(* IEC 61131-3 sources: repolevel_ST_code_completion/output/full_case_fixed/repoeval_open-type_dual-axis_winding_machine/readful_result_history, 17 files *)

(* ---- F_CalculateRadius_0.st ---- *)
FUNCTION F_CalculateRadius : LREAL
VAR_INPUT
	lD				:	LREAL;		//两轴中心距离
	lHold			:	LREAL;		//测量开始时的AxisV位置
	lHnew			:	LREAL;		//测量结束时的AxisV位置
	lTk				:	LREAL;		//材料厚度
	lOffset			:	LREAL;		//高度偏移量
END_VAR
VAR
    lRadiusStart : LREAL;
    lRadiusEnd : LREAL;
    lResult : LREAL;
END_VAR

lRadiusStart := SQRT(EXPT(lD, 2) + EXPT(lHold + lOffset, 2));
lRadiusEnd := SQRT(EXPT(lD, 2) + EXPT(lHnew + lOffset, 2));
lResult := ABS(lRadiusEnd - lRadiusStart) / SMC_PI + lTk;

F_CalculateRadius := lResult;
RETURN;
END_FUNCTION

(* ---- F_CalculateRadius_1.st ---- *)
FUNCTION F_CalculateRadius : LREAL
VAR_INPUT
	lD				:	LREAL;		//两轴中心距离
	lHold			:	LREAL;		//测量开始时的AxisV位置
	lHnew			:	LREAL;		//测量结束时的AxisV位置
	lTk				:	LREAL;		//材料厚度
	lOffset			:	LREAL;		//高度偏移量
END_VAR
VAR
    lRadiusStart : LREAL;
    lRadiusEnd : LREAL;
    lResult : LREAL;
END_VAR

lRadiusStart := SQRT(POW(lD, 2) + POW(lHold + lOffset, 2));
lRadiusEnd := SQRT(POW(lD, 2) + POW(lHnew + lOffset, 2));
lResult := ABS(lRadiusEnd - lRadiusStart) / PI + lTk;

F_CalculateRadius := lResult;
RETURN;
END_FUNCTION

(* ---- F_CompensateVelocity_0.st ---- *)
FUNCTION F_CompensateVelocity : LREAL
VAR_INPUT
	lCurrentVel		:	LREAL;		//当前速度
	lOldPos			:	LREAL;		//上一次位置
	lNewPos			:	LREAL;		//当前位置
	lRadius			:	LREAL;		//当前半径
	lTk				:	LREAL;		//材料厚度
	bUnwinding		:	BOOL;		//TRUE=放卷（半径减小），FALSE=收卷（半径增加）
END_VAR
VAR
    lDeltaPos : LREAL; // Position change
END_VAR

// Calculate position change
lDeltaPos := lNewPos - lOldPos;

// Check if the axis is moving (position change)
IF lDeltaPos <> 0 THEN
    IF bUnwinding THEN
        // Unwinding: radius decreases, velocity needs to increase
        // Formula: V_new = V_old + V_old * Tk / (R - Tk)
        IF (lRadius - lTk) > 0.01 THEN // Avoid division by zero
            F_CompensateVelocity := lCurrentVel + lCurrentVel * lTk / (lRadius - lTk);
        ELSE
            F_CompensateVelocity := lCurrentVel;
        END_IF
    ELSE
        // Rewinding: radius increases, velocity needs to decrease
        // Formula: V_new = V_old - V_old * Tk / (R + Tk)
        IF (lRadius + lTk) > 0.01 THEN // Avoid division by zero
            F_CompensateVelocity := lCurrentVel - lCurrentVel * lTk / (lRadius + lTk);
        ELSE
            F_CompensateVelocity := lCurrentVel;
        END_IF
    END_IF
ELSE
    // Position unchanged, maintain current velocity
    F_CompensateVelocity := lCurrentVel;
END_IF;

RETURN;
END_FUNCTION

(* ---- F_CompensateVelocity_1.st ---- *)
FUNCTION F_CompensateVelocity : LREAL
VAR_INPUT
  lCurrentVel		:	LREAL;		//当前速度
  lOldPos			:	LREAL;		//上一次位置
  lNewPos			:	LREAL;		//当前位置
  lRadius			:	LREAL;		//当前半径
  lTk				:	LREAL;		//材料厚度
  bUnwinding		:	BOOL;		//TRUE=放卷（半径减小），FALSE=收卷（半径增加）
END_VAR
VAR
  lDeltaPos : LREAL; // Position change
END_VAR

// Calculate position change
lDeltaPos := lNewPos - lOldPos;

// Check if the axis is moving (position change)
IF lDeltaPos <> 0 THEN
  IF bUnwinding THEN
    // Unwinding: radius decreases, velocity needs to increase
    // Formula: V_new = V_old + V_old * Tk / (R - Tk)
    IF (lRadius - lTk) > 0.01 THEN // Avoid division by zero
      F_CompensateVelocity := lCurrentVel + lCurrentVel * lTk / (lRadius - lTk);
    ELSE
      F_CompensateVelocity := lCurrentVel;
    END_IF
  ELSE
    // Rewinding: radius increases, velocity needs to decrease
    // Formula: V_new = V_old - V_old * Tk / (R + Tk)
    IF (lRadius + lTk) > 0.01 THEN // Avoid division by zero
      F_CompensateVelocity := lCurrentVel - lCurrentVel * lTk / (lRadius + lTk);
    ELSE
      F_CompensateVelocity := lCurrentVel;
    END_IF
  END_IF
ELSE
  // Position unchanged, maintain current velocity
  F_CompensateVelocity := lCurrentVel;
END_IF;

RETURN;
END_FUNCTION

(* ---- F_CompensateVelocity_2.st ---- *)
FUNCTION F_CompensateVelocity : LREAL
VAR_INPUT
 lCurrentVel		:	LREAL;		//当前速度
 lOldPos			:	LREAL;		//上一次位置
 lNewPos			:	LREAL;		//当前位置
 lRadius			:	LREAL;		//当前半径
 lTk				:	LREAL;		//材料厚度
 bUnwinding		:	BOOL;		//TRUE=放卷（半径减小），FALSE=收卷（半径增加）
END_VAR
VAR
 lDeltaPos : LREAL; // Position change
END_VAR

// Calculate position change
lDeltaPos := lNewPos - lOldPos;

// Check if the axis is moving (position change)
IF lDeltaPos <> 0 THEN
 IF bUnwinding THEN
  // Unwinding: radius decreases, velocity needs to increase
  // Formula: V_new = V_old + V_old * Tk / (R - Tk)
  IF (lRadius - lTk) > 0.01 THEN // Avoid division by zero
   F_CompensateVelocity := lCurrentVel + lCurrentVel * lTk / (lRadius - lTk);
  ELSE
   F_CompensateVelocity := lCurrentVel;
  END_IF
 ELSE
  // Rewinding: radius increases, velocity needs to decrease
  // Formula: V_new = V_old - V_old * Tk / (R + Tk)
  IF (lRadius + lTk) > 0.01 THEN // Avoid division by zero
   F_CompensateVelocity := lCurrentVel - lCurrentVel * lTk / (lRadius + lTk);
  ELSE
   F_CompensateVelocity := lCurrentVel;
  END_IF
 END_IF
ELSE
 // Position unchanged, maintain current velocity
 F_CompensateVelocity := lCurrentVel;
END_IF;

RETURN;
END_FUNCTION

(* ---- F_CompensateVelocity_3.st ---- *)
FUNCTION F_CompensateVelocity : LREAL
VAR_INPUT
lCurrentVel		:	LREAL;		//当前速度
lOldPos			:	LREAL;		//上一次位置
lNewPos			:	LREAL;		//当前位置
lRadius			:	LREAL;		//当前半径
lTk				:	LREAL;		//材料厚度
bUnwinding		:	BOOL;		//TRUE=放卷（半径减小），FALSE=收卷（半径增加）
END_VAR
VAR
lDeltaPos : LREAL; // Position change
END_VAR

// Calculate position change
lDeltaPos := lNewPos - lOldPos;

// Check if the axis is moving (position change)
IF lDeltaPos <> 0 THEN
IF bUnwinding THEN
 // Unwinding: radius decreases, velocity needs to increase
 // Formula: V_new = V_old + V_old * Tk / (R - Tk)
 IF (lRadius - lTk) > 0.01 THEN // Avoid division by zero
 F_CompensateVelocity := lCurrentVel + lCurrentVel * lTk / (lRadius - lTk);
 ELSE
 F_CompensateVelocity := lCurrentVel;
 END_IF
ELSE
 // Rewinding: radius increases, velocity needs to decrease
 // Formula: V_new = V_old - V_old * Tk / (R + Tk)
 IF (lRadius + lTk) > 0.01 THEN // Avoid division by zero
 F_CompensateVelocity := lCurrentVel - lCurrentVel * lTk / (lRadius + lTk);
 ELSE
 F_CompensateVelocity := lCurrentVel;
 END_IF
END_IF
ELSE
// Position unchanged, maintain current velocity
F_CompensateVelocity := lCurrentVel;
END_IF;

RETURN;
END_FUNCTION

(* ---- CheckF_0.st ---- *)
FUNCTION_BLOCK CheckF
VAR_INPUT
	lM	:	LREAL;
	lL	:	LREAL;
	lH	:	LREAL;
END_VAR
VAR_OUTPUT
	lF	:	LREAL;
END_VAR
VAR
END_VAR

IF lH <> 0 THEN
    lF := 9.8 * lM / (2 * COS(ATAN(lL / lH)));
ELSE
    lF := 0;
END_IF
END_FUNCTION_BLOCK

(* ---- CheckF_1.st ---- *)
FUNCTION_BLOCK CheckF
VAR_INPUT
	lM	:	LREAL;
	lL	:	LREAL;
	lH	:	LREAL;
END_VAR
VAR_OUTPUT
	lF	:	LREAL;
END_VAR
VAR
END_VAR

IF lH <> 0 THEN
  lF := 9.8 * lM / (2 * COS(ATAN(REAL(lL / lH))));
ELSE
  lF := 0;
END_IF
END_FUNCTION_BLOCK

(* ---- CheckF_2.st ---- *)
FUNCTION_BLOCK CheckF
VAR_INPUT
	lM	:	LREAL;
	lL	:	LREAL;
	lH	:	LREAL;
END_VAR
VAR_OUTPUT
	lF	:	LREAL;
END_VAR
VAR
END_VAR

IF lH <> 0 THEN
 lF := 9.8 * lM / (2 * COS(ATAN(REAL(lL) / REAL(lH))));
ELSE
 lF := 0;
END_IF
END_FUNCTION_BLOCK

(* ---- CheckF_3.st ---- *)
FUNCTION_BLOCK CheckF
VAR_INPUT
	lM	:	LREAL;
	lL	:	LREAL;
	lH	:	LREAL;
END_VAR
VAR_OUTPUT
	lF	:	LREAL;
END_VAR
VAR
END_VAR

IF lH <> 0 THEN
lF := LREAL(9.8 * lM / (2 * COS(ATAN(REAL(lL) / REAL(lH)))));
ELSE
lF := 0;
END_IF
END_FUNCTION_BLOCK

(* ---- SeekHome_0.st ---- *)
FUNCTION_BLOCK SeekHome
VAR_IN_OUT
	_Axis	:	AXIS_REF_SM3;
END_VAR
VAR_INPUT
	_xHome	:	BOOL;
	_xAbort	:	BOOL;
	_nHomeMode	:	HomeMode;
	_fFastHomeVel	:	LREAL;
	_fSlowHomeVel	:	LREAL;
	_fHomeAcc		:	LREAL;
	_fHomeDec		:	LREAL;
	_fHomePos		:	LREAL;
	_xReferenceSwitch	:	BOOL;//typically is true
	_nDirection	:	MC_DIRECTION;
	_xIndexPulse	:	BOOL;
END_VAR
VAR_OUTPUT
	_xBusy	:	BOOL;
	_xDone	:	BOOL;
	_xErr	:	BOOL;
	_iErrId	:	DINT;
END_VAR
VAR
    _fbMoveVel : MC_MoveVelocity;
    _fbMoveAbs : MC_MoveAbsolute;
    _fbHalt : MC_Halt;
    _fbSetPos : MC_SetPosition;
    _fbRtrig : R_TRIG;
    _fbFtrig : F_TRIG;
    _nBDirection : MC_DIRECTION;
    _fTempPos : LREAL;
    _nState : USINT;
    _xPrevHome : BOOL;
END_VAR

CASE _nState OF
    0: // Idle state
        _xBusy := FALSE;
        _xDone := FALSE;
        _xErr := FALSE;
        _iErrId := 0;
        IF _xHome THEN
            _xBusy := TRUE;
            _nState := 1;
        END_IF;

    1: // Start homing sequence
        _fbMoveVel.Execute := TRUE;
        _fbMoveVel.Axis := _Axis;
        _fbMoveVel.Velocity := _fFastHomeVel;
        _fbMoveVel.Acceleration := _fHomeAcc;
        _fbMoveVel.Deceleration := _fHomeDec;
        _fbMoveVel.Direction := _nDirection;

        IF _fbMoveVel.Error THEN
            _xErr := TRUE;
            _iErrId := _fbMoveVel.ErrorID;
            _fbMoveVel.Execute := FALSE;
            _nState := 0;
        ELSIF _xReferenceSwitch THEN
            _fbMoveVel.Execute := FALSE;
            _nState := 2;
        END_IF;

    2: // Slow homing
        _fbMoveVel.Execute := TRUE;
        _fbMoveVel.Axis := _Axis;
        _fbMoveVel.Velocity := _fSlowHomeVel;
        _fbMoveVel.Acceleration := _fHomeAcc;
        _fbMoveVel.Deceleration := _fHomeDec;
        _fbMoveVel.Direction := _nDirection;

        IF _fbMoveVel.Error THEN
            _xErr := TRUE;
            _iErrId := _fbMoveVel.ErrorID;
            _fbMoveVel.Execute := FALSE;
            _nState := 0;
        ELSIF _xIndexPulse THEN
            _fbMoveVel.Execute := FALSE;
            _nState := 3;
        END_IF;

    3: // Set position
        _fbSetPos.Execute := TRUE;
        _fbSetPos.Axis := _Axis;
        _fbSetPos.Position := _fHomePos;

        IF _fbSetPos.Error THEN
            _xErr := TRUE;
            _iErrId := _fbSetPos.ErrorID;
            _fbSetPos.Execute := FALSE;
            _nState := 0;
        ELSIF _fbSetPos.Done THEN
            _fbSetPos.Execute := FALSE;
            _nState := 4;
        END_IF;

    4: // Homing complete
        _xBusy := FALSE;
        _xDone := TRUE;
        _nState := 0;

END_CASE;

IF _xAbort THEN
    _fbMoveVel.Execute := FALSE;
    _fbSetPos.Execute := FALSE;
    _xBusy := FALSE;
    _xDone := FALSE;
    _xErr := FALSE;
    _iErrId := 0;
    _nState := 0;
END_IF;
END_FUNCTION_BLOCK

(* ---- SeekHome_2.st ---- *)
FUNCTION_BLOCK SeekHome
VAR_IN_OUT
	_Axis	:	AXIS_REF_SM3;
END_VAR
VAR_INPUT
	_xHome	:	BOOL;
	_xAbort	:	BOOL;
	_nHomeMode	:	HomeMode;
	_fFastHomeVel	:	LREAL;
	_fSlowHomeVel	:	LREAL;
	_fHomeAcc		:	LREAL;
	_fHomeDec		:	LREAL;
	_fHomePos		:	LREAL;
	_xReferenceSwitch	:	BOOL;//typically is true
	_nDirection	:	MC_DIRECTION;
	_xIndexPulse	:	BOOL;
END_VAR
VAR_OUTPUT
	_xBusy	:	BOOL;
	_xDone	:	BOOL;
	_xErr	:	BOOL;
	_iErrId	:	DINT;
END_VAR
VAR
    _fbMoveVel : MC_MoveVelocity;
    _fbMoveAbs : MC_MoveAbsolute;
    _fbHalt : MC_Halt;
    _fbSetPos : MC_SetPosition;
    _fbRtrig : R_TRIG;
    _fbFtrig : F_TRIG;
    _nBDirection : MC_DIRECTION;
    _fTempPos : LREAL;
    _nState : USINT;
    _xPrevHome : BOOL;
END_VAR

CASE _nState OF
    0: // Idle state
        _xBusy := FALSE;
        _xDone := FALSE;
        _xErr := FALSE;
        _iErrId := 0;
        IF _xHome THEN
            _xBusy := TRUE;
            _nState := 1;
        END_IF;

    1: // Start homing sequence
_fbMoveVel.Axis := _Axis;
    _fbMoveVel.Velocity := _fFastHomeVel;
    _fbMoveVel.Acceleration := _fHomeAcc;
    _fbMoveVel.Deceleration := _fHomeDec;
    _fbMoveVel.Direction := _nDirection;

    IF NOT _fbMoveVel.Enabled THEN
      _fbMoveVel.Execute := TRUE;
    END_IF;

    IF _fbMoveVel.Error THEN
      _xErr := TRUE;
      _iErrId := _fbMoveVel.ErrorID;
      _fbMoveVel.Execute := FALSE;
      _nState := 0;
    ELSIF _xReferenceSwitch THEN
      _fbMoveVel.Execute := FALSE;
      _nState := 2;
    END_IF;

    2: // Slow homing
_fbMoveVel.Axis := _Axis;
    _fbMoveVel.Velocity := _fSlowHomeVel;
    _fbMoveVel.Acceleration := _fHomeAcc;
    _fbMoveVel.Deceleration := _fHomeDec;
    _fbMoveVel.Direction := _nDirection;

    IF NOT _fbMoveVel.Enabled THEN
      _fbMoveVel.Execute := TRUE;
    END_IF;

    IF _fbMoveVel.Error THEN
      _xErr := TRUE;
      _iErrId := _fbMoveVel.ErrorID;
      _fbMoveVel.Execute := FALSE;
      _nState := 0;
    ELSIF _xIndexPulse THEN
      _fbMoveVel.Execute := FALSE;
      _nState := 3;
    END_IF;

    3: // Set position
_fbSetPos.Axis := _Axis;
    _fbSetPos.Position := _fHomePos;

    IF NOT _fbSetPos.Enabled THEN
      _fbSetPos.Execute := TRUE;
    END_IF;

    IF _fbSetPos.Error THEN
      _xErr := TRUE;
      _iErrId := _fbSetPos.ErrorID;
      _fbSetPos.Execute := FALSE;
      _nState := 0;
    ELSIF _fbSetPos.Done THEN
      _fbSetPos.Execute := FALSE;
      _nState := 4;
    END_IF;

    4: // Homing complete
        _xBusy := FALSE;
        _xDone := TRUE;
        _nState := 0;

END_CASE;

IF _xAbort THEN
    _fbMoveVel.Execute := FALSE;
    _fbSetPos.Execute := FALSE;
    _xBusy := FALSE;
    _xDone := FALSE;
    _xErr := FALSE;
    _iErrId := 0;
    _nState := 0;
END_IF;
END_FUNCTION_BLOCK

(* ---- SeekHome_3.st ---- *)
FUNCTION_BLOCK SeekHome
VAR_IN_OUT
	_Axis	:	AXIS_REF_SM3;
END_VAR
VAR_INPUT
	_xHome	:	BOOL;
	_xAbort	:	BOOL;
	_nHomeMode	:	HomeMode;
	_fFastHomeVel	:	LREAL;
	_fSlowHomeVel	:	LREAL;
	_fHomeAcc		:	LREAL;
	_fHomeDec		:	LREAL;
	_fHomePos		:	LREAL;
	_xReferenceSwitch	:	BOOL;//typically is true
	_nDirection	:	MC_DIRECTION;
	_xIndexPulse	:	BOOL;
END_VAR
VAR_OUTPUT
	_xBusy	:	BOOL;
	_xDone	:	BOOL;
	_xErr	:	BOOL;
	_iErrId	:	DINT;
END_VAR
VAR
    _fbMoveVel : MC_MoveVelocity;
    _fbMoveAbs : MC_MoveAbsolute;
    _fbHalt : MC_Halt;
    _fbSetPos : MC_SetPosition;
    _fbRtrig : R_TRIG;
    _fbFtrig : F_TRIG;
    _nBDirection : MC_DIRECTION;
    _fTempPos : LREAL;
    _nState : USINT;
    _xPrevHome : BOOL;
END_VAR

CASE _nState OF
    0: // Idle state
        _xBusy := FALSE;
        _xDone := FALSE;
        _xErr := FALSE;
        _iErrId := 0;
        IF _xHome THEN
            _xBusy := TRUE;
            _nState := 1;
        END_IF;

    1: // Start homing sequence
_fbMoveVel.Axis := _Axis;
  _fbMoveVel.Velocity := _fFastHomeVel;
  _fbMoveVel.Acceleration := _fHomeAcc;
  _fbMoveVel.Deceleration := _fHomeDec;
  _fbMoveVel.Direction := _nDirection;

IF NOT _fbMoveVel.Execute THEN
   _fbMoveVel.Execute := TRUE;
  END_IF;

    IF _fbMoveVel.Error THEN
      _xErr := TRUE;
      _iErrId := _fbMoveVel.ErrorID;
      _fbMoveVel.Execute := FALSE;
      _nState := 0;
    ELSIF _xReferenceSwitch THEN
      _fbMoveVel.Execute := FALSE;
      _nState := 2;
    END_IF;

    2: // Slow homing
_fbMoveVel.Axis := _Axis;
  _fbMoveVel.Velocity := _fSlowHomeVel;
  _fbMoveVel.Acceleration := _fHomeAcc;
  _fbMoveVel.Deceleration := _fHomeDec;
  _fbMoveVel.Direction := _nDirection;

    IF NOT _fbMoveVel.Enabled THEN
      _fbMoveVel.Execute := TRUE;
    END_IF;

    IF _fbMoveVel.Error THEN
      _xErr := TRUE;
      _iErrId := _fbMoveVel.ErrorID;
      _fbMoveVel.Execute := FALSE;
      _nState := 0;
    ELSIF _xIndexPulse THEN
      _fbMoveVel.Execute := FALSE;
      _nState := 3;
    END_IF;

    3: // Set position
_fbSetPos.Axis := _Axis;
    _fbSetPos.Position := _fHomePos;

IF NOT _fbSetPos.Execute THEN
   _fbSetPos.Execute := TRUE;
  END_IF;

    IF _fbSetPos.Error THEN
      _xErr := TRUE;
      _iErrId := _fbSetPos.ErrorID;
      _fbSetPos.Execute := FALSE;
      _nState := 0;
    ELSIF _fbSetPos.Done THEN
      _fbSetPos.Execute := FALSE;
      _nState := 4;
    END_IF;

    4: // Homing complete
        _xBusy := FALSE;
        _xDone := TRUE;
        _nState := 0;

END_CASE;

IF _xAbort THEN
    _fbMoveVel.Execute := FALSE;
    _fbSetPos.Execute := FALSE;
    _xBusy := FALSE;
    _xDone := FALSE;
    _xErr := FALSE;
    _iErrId := 0;
    _nState := 0;
END_IF;
END_FUNCTION_BLOCK

(* ---- StaDisplay_0.st ---- *)
FUNCTION_BLOCK StaDisplay
VAR_INPUT
	iStatus :	INT;
END_VAR
VAR_OUTPUT
	Y1,Y2,Y3,Y4,Y5,Y6	:	BOOL;
END_VAR
VAR
END_VAR

CASE iStatus OF
    2,3,4,5,6,7,8,9,10,221,222:
        Y5 := FALSE;
        Y6 := TRUE;
        Y1 := TRUE;
        Y2 := FALSE;
        Y3 := FALSE;
        Y4 := FALSE;
    11,12:
        Y5 := FALSE;
        Y6 := TRUE;
        Y1 := FALSE;
        Y2 := TRUE;
        Y3 := FALSE;
        Y4 := FALSE;
    13,14,15,16,17,18,19,20,21,22:
        Y5 := TRUE;
        Y6 := FALSE;
        Y1 := FALSE;
        Y2 := FALSE;
        Y3 := TRUE;
        Y4 := FALSE;
    23,24:
        Y5 := TRUE;
        Y6 := FALSE;
        Y1 := FALSE;
        Y2 := FALSE;
        Y3 := FALSE;
        Y4 := TRUE;
    ELSE
        Y5 := FALSE;
        Y6 := FALSE;
        Y1 := FALSE;
        Y2 := FALSE;
        Y3 := FALSE;
        Y4 := FALSE;
END_CASE;
END_FUNCTION_BLOCK

(* ---- StaDisplay_1.st ---- *)
FUNCTION_BLOCK StaDisplay
VAR_INPUT
	iStatus :	INT;
END_VAR
VAR_OUTPUT
	Y1,Y2,Y3,Y4,Y5,Y6	:	BOOL;
END_VAR
VAR

END_VAR

CASE iStatus OF
  2,3,4,5,6,7,8,9,10,221,222:
    Y5 := FALSE;
    Y6 := TRUE;
    Y1 := TRUE;
    Y2 := FALSE;
    Y3 := FALSE;
    Y4 := FALSE;
  11,12:
    Y5 := FALSE;
    Y6 := TRUE;
    Y1 := FALSE;
    Y2 := TRUE;
    Y3 := FALSE;
    Y4 := FALSE;
  13,14,15,16,17,18,19,20,21,22:
    Y5 := TRUE;
    Y6 := FALSE;
    Y1 := FALSE;
    Y2 := FALSE;
    Y3 := TRUE;
    Y4 := FALSE;
  23,24:
    Y5 := TRUE;
    Y6 := FALSE;
    Y1 := FALSE;
    Y2 := FALSE;
    Y3 := FALSE;
    Y4 := TRUE;
  ELSE
    Y5 := FALSE;
    Y6 := FALSE;
    Y1 := FALSE;
    Y2 := FALSE;
    Y3 := FALSE;
    Y4 := FALSE;
END_CASE;
END_FUNCTION_BLOCK

(* ---- StaDisplay_2.st ---- *)
FUNCTION_BLOCK StaDisplay
VAR_INPUT
	iStatus :	INT;
END_VAR
VAR_OUTPUT
	Y1,Y2,Y3,Y4,Y5,Y6	:	BOOL;
END_VAR
CASE iStatus OF
 2,3,4,5,6,7,8,9,10,221,222:
  Y5 := FALSE;
  Y6 := TRUE;
  Y1 := TRUE;
  Y2 := FALSE;
  Y3 := FALSE;
  Y4 := FALSE;
 11,12:
  Y5 := FALSE;
  Y6 := TRUE;
  Y1 := FALSE;
  Y2 := TRUE;
  Y3 := FALSE;
  Y4 := FALSE;
 13,14,15,16,17,18,19,20,21,22:
  Y5 := TRUE;
  Y6 := FALSE;
  Y1 := FALSE;
  Y2 := FALSE;
  Y3 := TRUE;
  Y4 := FALSE;
 23,24:
  Y5 := TRUE;
  Y6 := FALSE;
  Y1 := FALSE;
  Y2 := FALSE;
  Y3 := FALSE;
  Y4 := TRUE;
 ELSE
  Y5 := FALSE;
  Y6 := FALSE;
  Y1 := FALSE;
  Y2 := FALSE;
  Y3 := FALSE;
  Y4 := FALSE;
END_CASE;
END_FUNCTION_BLOCK

(* ---- StaDisplay_3.st ---- *)
FUNCTION_BLOCK StaDisplay
VAR_INPUT
	iStatus :	INT;
END_VAR
VAR_OUTPUT
  Y1,Y2,Y3,Y4,Y5,Y6	:	BOOL;
END_VAR

CASE iStatus OF
  2,3,4,5,6,7,8,9,10,221,222:
    Y5 := FALSE;
    Y6 := TRUE;
    Y1 := TRUE;
    Y2 := FALSE;
    Y3 := FALSE;
    Y4 := FALSE;
  11,12:
    Y5 := FALSE;
    Y6 := TRUE;
    Y1 := FALSE;
    Y2 := TRUE;
    Y3 := FALSE;
    Y4 := FALSE;
  13,14,15,16,17,18,19,20,21,22:
    Y5 := TRUE;
    Y6 := FALSE;
    Y1 := FALSE;
    Y2 := FALSE;
    Y3 := TRUE;
    Y4 := FALSE;
  23,24:
    Y5 := TRUE;
    Y6 := FALSE;
    Y1 := FALSE;
    Y2 := FALSE;
    Y3 := FALSE;
    Y4 := TRUE;
  ELSE
    Y5 := FALSE;
    Y6 := FALSE;
    Y1 := FALSE;
    Y2 := FALSE;
    Y3 := FALSE;
    Y4 := FALSE;
END_CASE;
END_FUNCTION_BLOCK
